TYPE
    Coordinates :
    STRUCT
        xValue        : DINT;
        yValue        : DINT;
        variableValue : DINT;
    END_STRUCT
END_TYPE

(* stored: Version 1.1.0.1, ProductVersion 3.1.4024.12
   DUT Coordinates: Id {ecab6d85-6b52-00f4-35bb-82c8c8bcef08} *)
